# EPICS substitutions: app/Db/ict.substitutions
file ictPdu.template
{
	{
		FOO = "whatever"
	}
}
